KUKA KRL data list: up112.dat

&ACCESS RVP
&REL 2
&COMMENT Wartung Greifer 1 VW380
&PARAM DISKPATH = UPs
&PARAM TEMPLATE = C:\KRC\Roboter\Template\upvorgabe
&PARAM TPVW_VERSION = 8.1.8
&PARAM EDITMASK = Up999[1-999]
DEFDAT UP112
; FOLD ;%{H} %MKUKATPVW
; ENDFOLD
; interface to basic routines
 EXT  BAS (BAS_COMMAND  :IN,REAL  :IN )
; interface to VW-standard routines
EXT VW (VW_COMMAND:IN, BOOL: IN, REAL:IN, REAL:IN, REAL:IN, REAL:IN, BOOL :IN, E6POS :IN )
; interface to VW_USER - Call
EXT  VW_USER (VW_USER_CMD :IN,INT :IN,REAL  :IN,REAL  :IN,REAL  :IN,REAL  :IN,REAL  :IN,REAL  :IN,BOOL  :IN )
EXT  VW_USR_R (VW_USER_CMD :IN,INT :IN,REAL  :IN,REAL  :IN,REAL  :IN,REAL  :IN,REAL  :IN,REAL  :IN,BOOL  :IN )
EXT  IBGN (IBGN_COMMAND  :IN,BOOL  :IN,REAL  :IN,REAL  :IN,BOOL  :IN,E6POS  :OUT )
; interface select routine
EXTFCT INT  SELECT (SUBTYPE  :IN,INT  :IN,BOOL  :IN,ARI_TYP  :IN,INT  :IN,BOOL_TYP  :IN,INT  :IN,BOOL  :IN)
INT VW_NEXT_FREE = 6
INT VW_NFREE_SPS = 6
INT VW_MAX_SPS = 106
DECL VW_MPARA_TYP P1_D = {TOOL_NO 12,BASE_NO 0,VB 100,VE 0,ACC 100,TRG_TIME 0,MOVE_TYPE #PTP_MOTION}
DECL E6POS P1 = {X 1644.416, Y -174.6792, Z 2340.625, A 0.01452038, B 29.99903, C -90.35256, S 2, T 42 , E1 0.0, E2 0.0, E3 0.0, E4 0.0, E5 0.0, E6 0.0}
DECL VW_MPARA_TYP P2_D = {TOOL_NO 12,BASE_NO 0,VB 100,VE 100,ACC 100,TRG_TIME 0,MOVE_TYPE #PTP_MOTION}
DECL E6POS P2 = {X 2388.61, Y -438.7298, Z 1083.309, A -2.522015, B 49.97304, C -8.240117, S 2, T 42 , E1 0.0, E2 0.0, E3 0.0, E4 0.0, E5 0.0, E6 0.0}
DECL VW_MPARA_TYP P3_D = {TOOL_NO 12,BASE_NO 0,VB 100,VE 0,ACC 100,TRG_TIME 5,MOVE_TYPE #PTP_MOTION}
DECL E6POS P3 = {X 2514.471, Y -762.2805, Z -712.819, A 4.802316, B 87.00743, C 6.317693, S 2, T 42 , E1 0.0, E2 0.0, E3 0.0, E4 0.0, E5 0.0, E6 0.0}
DECL VW_MPARA_TYP P4_D = {TOOL_NO 12,BASE_NO 0,VB 100,VE 100,ACC 100,TRG_TIME 0,MOVE_TYPE #PTP_MOTION}
DECL E6POS P4 = {X 2388.611, Y -438.729, Z 1083.309, A -2.522027, B 49.97306, C -8.240271, S 2, T 42 , E1 0.0, E2 0.0, E3 0.0, E4 0.0, E5 0.0, E6 0.0}
DECL VW_MPARA_TYP P5_D = {TOOL_NO 12,BASE_NO 0,VB 100,VE 0,ACC 100,TRG_TIME 0,MOVE_TYPE #PTP_MOTION}
DECL E6POS P5 = {X 1644.416, Y -174.6797, Z 2340.624, A 0.01450222, B 29.99903, C -90.35255, S 2, T 42 , E1 0.0, E2 0.0, E3 0.0, E4 0.0, E5 0.0, E6 0.0}
ENDDAT
